// SIMATIC S7-200 project (STEP 7-Micro/WIN), CPU 224XP CN REL 02.01

SYMBOL_TABLE Symbol Table
急停按钮             I0.0
水箱低液位保护          I0.1
量热器低液位保护         I0.2
循环泵水流开关          I0.3
低压保护             I0.4
高压保护             I0.5
高压开关             I0.6
压缩机箱机械温控         I0.7
变频器运行开关          I1.0
变频器故障开关          I1.1
防干烧1             I1.2
防干烧2             I1.3
UT1输出            Q0.0
UT2输出            Q0.1
UT3输出            Q0.2
UT4输出            Q0.3
UT5输出            Q0.4
UT6输出            Q0.5
供水泵              Q0.6
循环泵              Q0.7
压缩冷凝机组压缩机        Q1.0
压缩冷凝机组冷凝风机1      Q1.1
压缩冷凝机组冷凝风机2      Q2.0
压缩冷凝机组电磁阀        Q2.1
压缩冷凝机组加热器        Q2.2
水箱加热器            Q2.3
压缩机驱动电机          Q2.4
压缩机箱风机           Q2.5
压缩机机箱电加热器1       Q2.6
被测压缩冷凝机组         Q2.7
量热器加热器1          Q3.0
量热器加热器2          Q3.1
蜂鸣器报警            Q3.2
变频器运转            Q3.3
水路转换电磁阀          Q3.4
制冷剂路转换电磁阀1       Q3.5
制冷剂路转换电磁阀2       Q3.6
离合器              Q3.7
出口水温流量计转换UT4输    Q4.0
进口水温出水温度转换UT5    Q4.1
UT3UT4输出转换卡尔阀输   Q4.2
富士金电动调节阀供电       Q4.3
压缩机箱电加热器2        Q4.4
离合器DC24DC12切换    Q4.5
电机变频器故障          Q4.6
水箱液位报警           Q4.7
量热器液位报警          Q5.0
压缩机组报警           Q5.1
驱动电机报警           Q5.2
被测机组电磁阀          Q5.3
备用2              Q5.4
备用3              Q5.5
备用4              Q5.6
备用5              Q5.7
UT1输出继电器         M0.0
UT2输出继电          M0.1
UT3输出继电器         M0.2
UT4输出继电器         M0.3
UT5输出继电器         M0.4
UT6输出继电器         M0.5
供水泵继电器           M0.6
循环泵继电器           M0.7
压缩冷凝机组压缩机继电      M1.0
压缩冷凝机组冷凝风机1继     M1.1
低压保护软件寄存器        M1.2
急停寄存器            M1.3
防干烧1继电           M1.4
防干烧2继电           M1.5
蜂鸣器报警继电          M1.6
量热器报警            M1.7
压缩冷凝机组冷凝风机2继     M2.0
压缩冷凝机组电磁阀继电      M2.1
压缩冷凝机组加热器继电      M2.2
水箱加热器继电器         M2.3
压缩机驱动电机继电器       M2.4
压缩机箱风机继电器        M2.5
压缩机机箱电加热器1继电     M2.6
被测压缩冷凝机组继电器      M2.7
量热器加热器1继电器       M3.0
量热器加热器2继电器       M3.1
蜂鸣器报警继电器         M3.2
变频器运转继电器         M3.3
水路转换电磁阀继电器       M3.4
制冷剂路转换电磁阀1继电     M3.5
制冷剂路转换电磁阀2继电     M3.6
离合器继电器           M3.7
出口水温流量计UT4继电器    M4.0
进口出水温度转换UT5继     M4.1
UT3UT4输出转换继电器    M4.2
电动调节阀供电继电器       M4.3
压缩机箱电加热器2继电器     M4.4
离合器DC24DC12切换继电  M4.5
电机变频器故障继电        M4.6
水箱液位报警继电         M4.7
量热器液位报警继电        M5.0
压缩机组报警继电         M5.1
驱动电机报警继电         M5.2
被测机组电磁阀继电        M5.3
备用2继电            M5.4
备用3继电            M5.5
备用4继电            M5.6
备用5继电            M5.7
END_SYMBOL_TABLE

ORGANIZATION_BLOCK 主程序:OB1
TITLE=程序注释
BEGIN
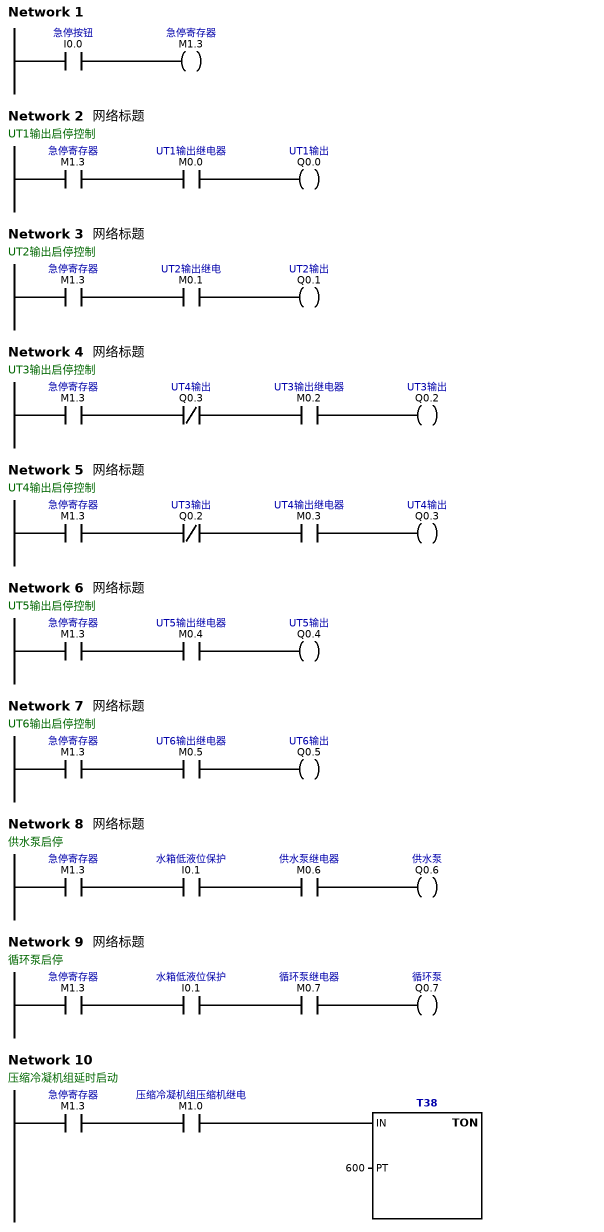
Network 1
LD     急停按钮:I0.0
=      急停寄存器:M1.3
Network 2 // 网络标题
// UT1输出启停控制
LD     急停寄存器:M1.3
A      UT1输出继电器:M0.0
=      UT1输出:Q0.0
Network 3 // 网络标题
// UT2输出启停控制
LD     急停寄存器:M1.3
A      UT2输出继电:M0.1
=      UT2输出:Q0.1
Network 4 // 网络标题
// UT3输出启停控制
LD     急停寄存器:M1.3
AN     UT4输出:Q0.3
A      UT3输出继电器:M0.2
=      UT3输出:Q0.2
Network 5 // 网络标题
// UT4输出启停控制
LD     急停寄存器:M1.3
AN     UT3输出:Q0.2
A      UT4输出继电器:M0.3
=      UT4输出:Q0.3
Network 6 // 网络标题
// UT5输出启停控制
LD     急停寄存器:M1.3
A      UT5输出继电器:M0.4
=      UT5输出:Q0.4
Network 7 // 网络标题
// UT6输出启停控制
LD     急停寄存器:M1.3
A      UT6输出继电器:M0.5
=      UT6输出:Q0.5
Network 8 // 网络标题
// 供水泵启停
LD     急停寄存器:M1.3
A      水箱低液位保护:I0.1
A      供水泵继电器:M0.6
=      供水泵:Q0.6
Network 9 // 网络标题
// 循环泵启停
LD     急停寄存器:M1.3
A      水箱低液位保护:I0.1
A      循环泵继电器:M0.7
=      循环泵:Q0.7
Network 10
// 压缩冷凝机组延时启动
LD     急停寄存器:M1.3
A      压缩冷凝机组压缩机继电:M1.0
TON    T38, 600
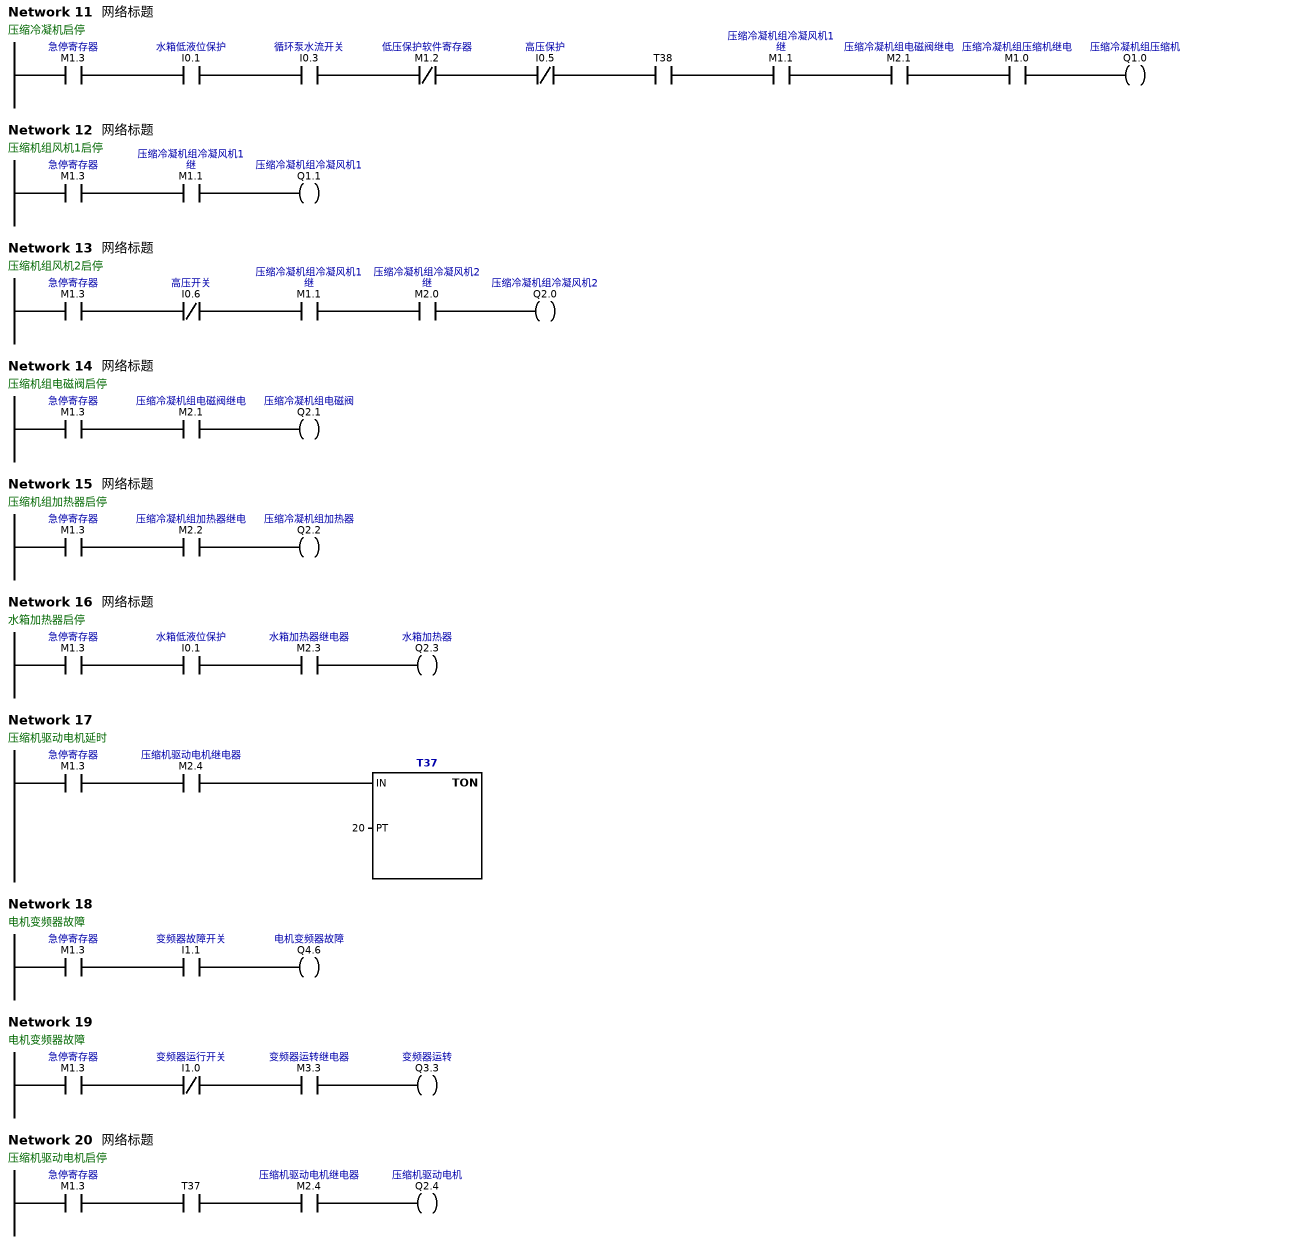
Network 11 // 网络标题
// 压缩冷凝机启停
LD     急停寄存器:M1.3
A      水箱低液位保护:I0.1
A      循环泵水流开关:I0.3
AN     低压保护软件寄存器:M1.2
AN     高压保护:I0.5
A      T38
A      压缩冷凝机组冷凝风机1继:M1.1
A      压缩冷凝机组电磁阀继电:M2.1
A      压缩冷凝机组压缩机继电:M1.0
=      压缩冷凝机组压缩机:Q1.0
Network 12 // 网络标题
// 压缩机组风机1启停
LD     急停寄存器:M1.3
A      压缩冷凝机组冷凝风机1继:M1.1
=      压缩冷凝机组冷凝风机1:Q1.1
Network 13 // 网络标题
// 压缩机组风机2启停
LD     急停寄存器:M1.3
AN     高压开关:I0.6
A      压缩冷凝机组冷凝风机1继:M1.1
A      压缩冷凝机组冷凝风机2继:M2.0
=      压缩冷凝机组冷凝风机2:Q2.0
Network 14 // 网络标题
// 压缩机组电磁阀启停
LD     急停寄存器:M1.3
A      压缩冷凝机组电磁阀继电:M2.1
=      压缩冷凝机组电磁阀:Q2.1
Network 15 // 网络标题
// 压缩机组加热器启停
LD     急停寄存器:M1.3
A      压缩冷凝机组加热器继电:M2.2
=      压缩冷凝机组加热器:Q2.2
Network 16 // 网络标题
// 水箱加热器启停
LD     急停寄存器:M1.3
A      水箱低液位保护:I0.1
A      水箱加热器继电器:M2.3
=      水箱加热器:Q2.3
Network 17
// 压缩机驱动电机延时
LD     急停寄存器:M1.3
A      压缩机驱动电机继电器:M2.4
TON    T37, 20
Network 18
// 电机变频器故障
LD     急停寄存器:M1.3
A      变频器故障开关:I1.1
=      电机变频器故障:Q4.6
Network 19
// 电机变频器故障
LD     急停寄存器:M1.3
AN     变频器运行开关:I1.0
A      变频器运转继电器:M3.3
=      变频器运转:Q3.3
Network 20 // 网络标题
// 压缩机驱动电机启停
LD     急停寄存器:M1.3
A      T37
A      压缩机驱动电机继电器:M2.4
=      压缩机驱动电机:Q2.4
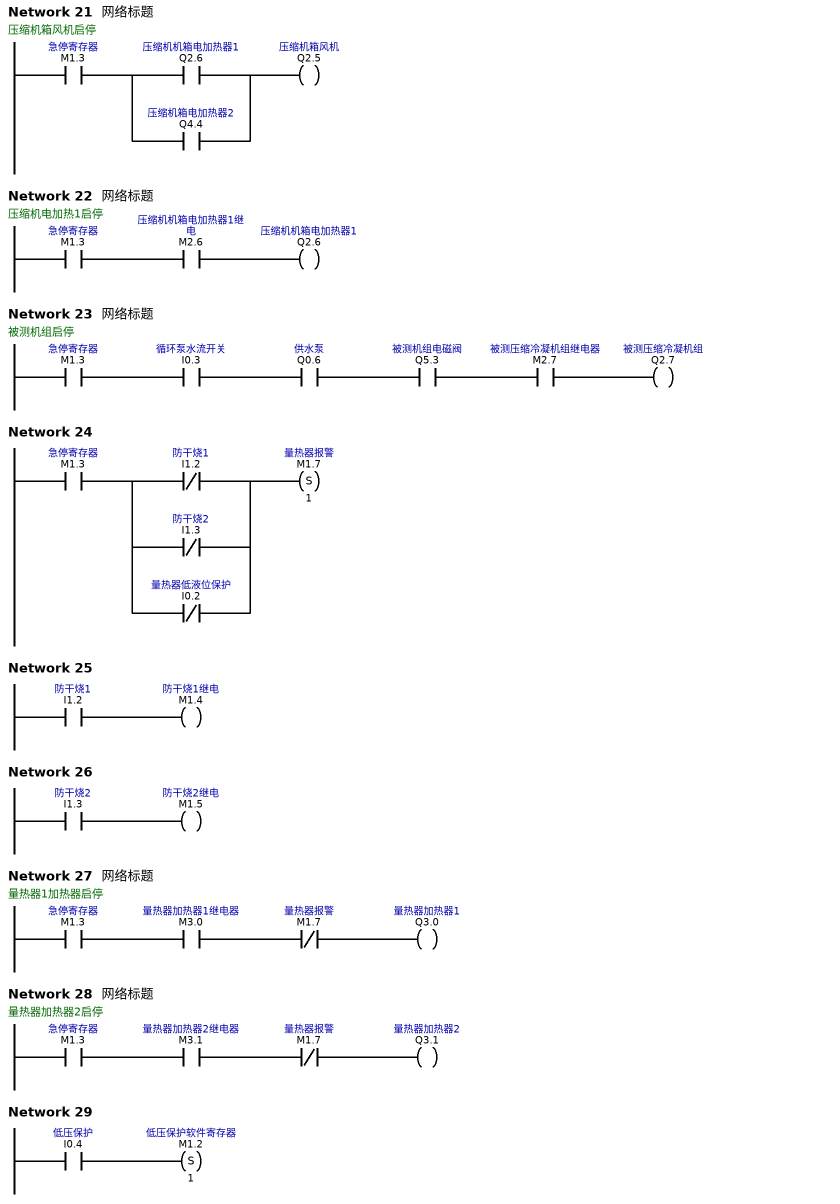
Network 21 // 网络标题
// 压缩机箱风机启停
LD     急停寄存器:M1.3
LD     压缩机机箱电加热器1:Q2.6
O      压缩机箱电加热器2:Q4.4
ALD
=      压缩机箱风机:Q2.5
Network 22 // 网络标题
// 压缩机电加热1启停
LD     急停寄存器:M1.3
A      压缩机机箱电加热器1继电:M2.6
=      压缩机机箱电加热器1:Q2.6
Network 23 // 网络标题
// 被测机组启停
LD     急停寄存器:M1.3
A      循环泵水流开关:I0.3
A      供水泵:Q0.6
A      被测机组电磁阀:Q5.3
A      被测压缩冷凝机组继电器:M2.7
=      被测压缩冷凝机组:Q2.7
Network 24
LD     急停寄存器:M1.3
LDN    防干烧1:I1.2
ON     防干烧2:I1.3
ON     量热器低液位保护:I0.2
ALD
S      量热器报警:M1.7, 1
Network 25
LD     防干烧1:I1.2
=      防干烧1继电:M1.4
Network 26
LD     防干烧2:I1.3
=      防干烧2继电:M1.5
Network 27 // 网络标题
// 量热器1加热器启停
LD     急停寄存器:M1.3
A      量热器加热器1继电器:M3.0
AN     量热器报警:M1.7
=      量热器加热器1:Q3.0
Network 28 // 网络标题
// 量热器加热器2启停
LD     急停寄存器:M1.3
A      量热器加热器2继电器:M3.1
AN     量热器报警:M1.7
=      量热器加热器2:Q3.1
Network 29
LD     低压保护:I0.4
S      低压保护软件寄存器:M1.2, 1
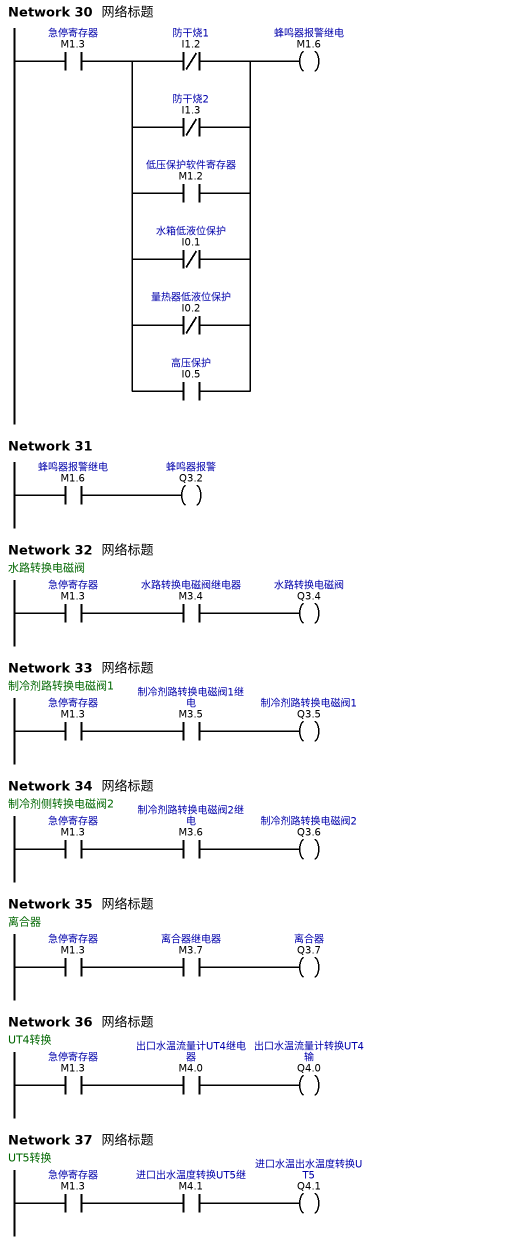
Network 30 // 网络标题
LD     急停寄存器:M1.3
LDN    防干烧1:I1.2
ON     防干烧2:I1.3
O      低压保护软件寄存器:M1.2
ON     水箱低液位保护:I0.1
ON     量热器低液位保护:I0.2
O      高压保护:I0.5
ALD
=      蜂鸣器报警继电:M1.6
Network 31
LD     蜂鸣器报警继电:M1.6
=      蜂鸣器报警:Q3.2
Network 32 // 网络标题
// 水路转换电磁阀
LD     急停寄存器:M1.3
A      水路转换电磁阀继电器:M3.4
=      水路转换电磁阀:Q3.4
Network 33 // 网络标题
// 制冷剂路转换电磁阀1
LD     急停寄存器:M1.3
A      制冷剂路转换电磁阀1继电:M3.5
=      制冷剂路转换电磁阀1:Q3.5
Network 34 // 网络标题
// 制冷剂侧转换电磁阀2
LD     急停寄存器:M1.3
A      制冷剂路转换电磁阀2继电:M3.6
=      制冷剂路转换电磁阀2:Q3.6
Network 35 // 网络标题
// 离合器
LD     急停寄存器:M1.3
A      离合器继电器:M3.7
=      离合器:Q3.7
Network 36 // 网络标题
// UT4转换
LD     急停寄存器:M1.3
A      出口水温流量计UT4继电器:M4.0
=      出口水温流量计转换UT4输:Q4.0
Network 37 // 网络标题
// UT5转换
LD     急停寄存器:M1.3
A      进口出水温度转换UT5继:M4.1
=      进口水温出水温度转换UT5:Q4.1
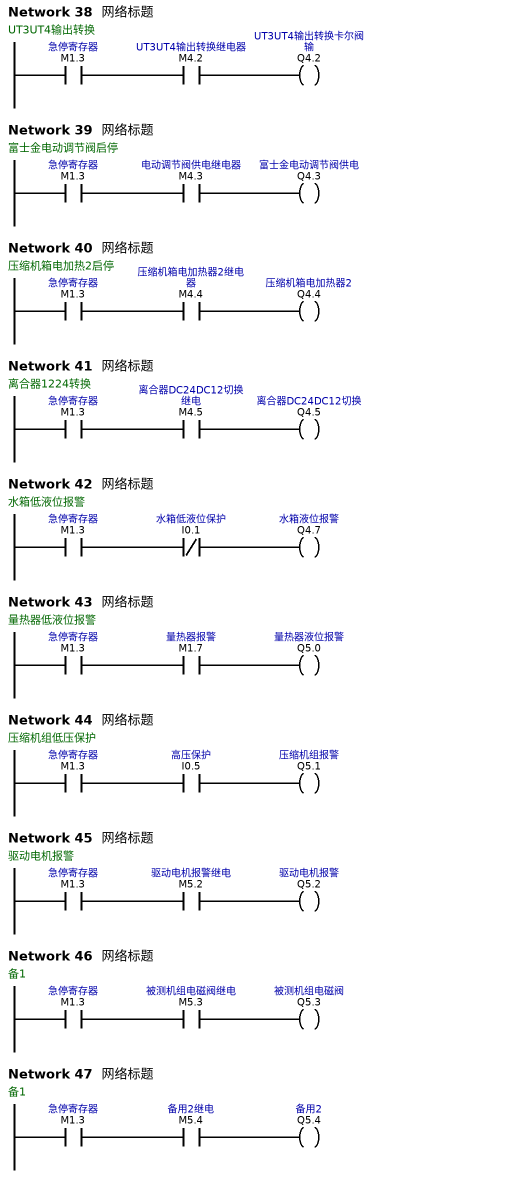
Network 38 // 网络标题
// UT3UT4输出转换
LD     急停寄存器:M1.3
A      UT3UT4输出转换继电器:M4.2
=      UT3UT4输出转换卡尔阀输:Q4.2
Network 39 // 网络标题
// 富士金电动调节阀启停
LD     急停寄存器:M1.3
A      电动调节阀供电继电器:M4.3
=      富士金电动调节阀供电:Q4.3
Network 40 // 网络标题
// 压缩机箱电加热2启停
LD     急停寄存器:M1.3
A      压缩机箱电加热器2继电器:M4.4
=      压缩机箱电加热器2:Q4.4
Network 41 // 网络标题
// 离合器1224转换
LD     急停寄存器:M1.3
A      离合器DC24DC12切换继电:M4.5
=      离合器DC24DC12切换:Q4.5
Network 42 // 网络标题
// 水箱低液位报警
LD     急停寄存器:M1.3
AN     水箱低液位保护:I0.1
=      水箱液位报警:Q4.7
Network 43 // 网络标题
// 量热器低液位报警
LD     急停寄存器:M1.3
A      量热器报警:M1.7
=      量热器液位报警:Q5.0
Network 44 // 网络标题
// 压缩机组低压保护
LD     急停寄存器:M1.3
A      高压保护:I0.5
=      压缩机组报警:Q5.1
Network 45 // 网络标题
// 驱动电机报警
LD     急停寄存器:M1.3
A      驱动电机报警继电:M5.2
=      驱动电机报警:Q5.2
Network 46 // 网络标题
// 备1
LD     急停寄存器:M1.3
A      被测机组电磁阀继电:M5.3
=      被测机组电磁阀:Q5.3
Network 47 // 网络标题
// 备1
LD     急停寄存器:M1.3
A      备用2继电:M5.4
=      备用2:Q5.4
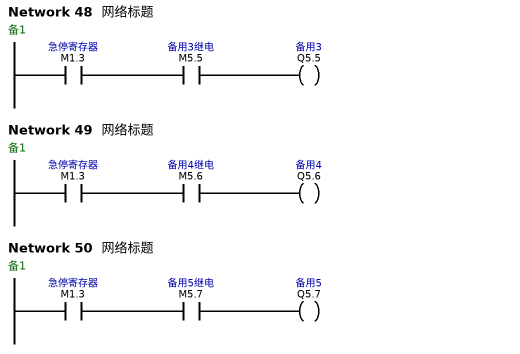
Network 48 // 网络标题
// 备1
LD     急停寄存器:M1.3
A      备用3继电:M5.5
=      备用3:Q5.5
Network 49 // 网络标题
// 备1
LD     急停寄存器:M1.3
A      备用4继电:M5.6
=      备用4:Q5.6
Network 50 // 网络标题
// 备1
LD     急停寄存器:M1.3
A      备用5继电:M5.7
=      备用5:Q5.7
END_ORGANIZATION_BLOCK
